SYSTEM OPC_Test
  (* Description: Showing how to use more than one forte on the same PC connection via OPC UA. One forte PC using as server, the other(s) as client(s). requirements: - one running forte PC on standard configuration - one running forte PC started on port 61599 ("-c localhost:61599") - OPC UA is required for all forte PCs *)
  (* Version 1.0, 2022-04-26, Maximilian Scharf *)
  APPLICATION OPC_TestApp
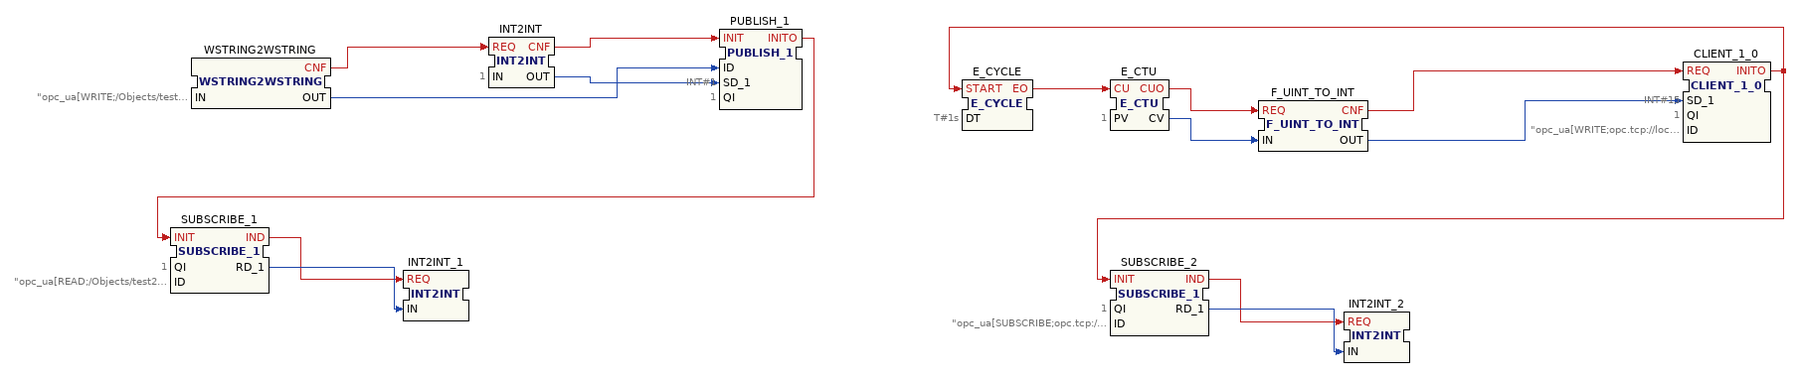
    (* Group __Group01: OPC UA documentation &#10;https://www.eclipse.org/4diac/en_help.php?helppage=html/communication/opc_ua_version1.html#build *)
    (* Group __Group02: OPC UA Server &#10;use: publish (WRITE) and subscribe (READ) *)
    (* Group __Group03: OPC UA Client &#10;use: client (WRITE) or subscribe (SUBSCRIBE) FBs *)
    (* Group __Group04: Use UaExpert Client for OPC UA connection and monitoring. *)
    FBS
      WSTRING2WSTRING : WSTRING2WSTRING(IN := "opc_ua[WRITE;/Objects/test1]"); {SET_ATTRIBUTE(GroupName, __Group02)}
      E_CTU : E_CTU(PV := 1); {SET_ATTRIBUTE(GroupName, __Group03)}
      E_CYCLE : E_CYCLE(DT := T#1s); {SET_ATTRIBUTE(GroupName, __Group03)}
      PUBLISH_1 : PUBLISH_1(QI := 1, SD_1 := INT#1); {SET_ATTRIBUTE(GroupName, __Group02)}
      CLIENT_1_0 : CLIENT_1_0(QI := 1, ID := "opc_ua[WRITE;opc.tcp://localhost:4840#;/Objects/test2]", SD_1 := INT#15); {SET_ATTRIBUTE(GroupName, __Group03)}
      INT2INT : INT2INT(IN := 1); {SET_ATTRIBUTE(GroupName, __Group02)}
      F_UINT_TO_INT : F_UINT_TO_INT; {SET_ATTRIBUTE(GroupName, __Group03)}
      SUBSCRIBE_1 : SUBSCRIBE_1(QI := 1, ID := "opc_ua[READ;/Objects/test2]"); {SET_ATTRIBUTE(GroupName, __Group02)}
      INT2INT_1 : INT2INT; {SET_ATTRIBUTE(GroupName, __Group02)}
      SUBSCRIBE_2 : SUBSCRIBE_1(QI := 1, ID := "opc_ua[SUBSCRIBE;opc.tcp://localhost:4840#;/Objects/test2]"); {SET_ATTRIBUTE(GroupName, __Group03)}
      INT2INT_2 : INT2INT; {SET_ATTRIBUTE(GroupName, __Group03)}
    END_FBS
    EVENT_CONNECTIONS
      E_CYCLE.EO TO E_CTU.CU;
      CLIENT_1_0.INITO TO E_CYCLE.START;
      INT2INT.CNF TO PUBLISH_1.INIT;
      WSTRING2WSTRING.CNF TO INT2INT.REQ;
      E_CTU.CUO TO F_UINT_TO_INT.REQ;
      F_UINT_TO_INT.CNF TO CLIENT_1_0.REQ;
      PUBLISH_1.INITO TO SUBSCRIBE_1.INIT;
      SUBSCRIBE_1.IND TO INT2INT_1.REQ;
      SUBSCRIBE_2.IND TO INT2INT_2.REQ;
      CLIENT_1_0.INITO TO SUBSCRIBE_2.INIT;
    END_CONNECTIONS
    DATA_CONNECTIONS
      WSTRING2WSTRING.OUT TO PUBLISH_1.ID;
      INT2INT.OUT TO PUBLISH_1.SD_1;
      E_CTU.CV TO F_UINT_TO_INT.IN;
      F_UINT_TO_INT.OUT TO CLIENT_1_0.SD_1;
      SUBSCRIBE_1.RD_1 TO INT2INT_1.IN;
      SUBSCRIBE_2.RD_1 TO INT2INT_2.IN;
    END_CONNECTIONS
  END_APPLICATION
  DEVICE Server : FORTE_PC(MGR_ID := "localhost:61498")
    {SET_ATTRIBUTE(Profile, DynamicTypeLoad)}
    {SET_ATTRIBUTE(FBType, GEN_E_MUX, F_LT, F_LWORD_TO_WORD, F_TAN, F_DINT_TO_UINT, F_BYTE_TO_DINT, F_ADD_DT_TIME, F_TIME_IN_US_TO_LREAL, F_INT_TO_UDINT, F_ADD_TOD_TIME, F_SUB_DT_DT, F_DT_TO_TOD, F_WSTRING_TO_REAL, F_UINT_TO_BCD_WORD, F_UDINT_TO_REAL, F_REAL_TO_UDINT, F_DWORD_TO_WORD, F_MUL, FB_CTUD_LINT, TEST_CONDITION, F_LE, GEN_SUBSCRIBE, F_LN, FB_CTD_DINT, GEN_OR, E_CYCLE, FB_F_TRIG, F_LREAL_TO_SINT, E_F_TRIG, F_LWORD_TO_UINT, E_RS, F_UINT_TO_WORD, F_WORD_TO_DINT, F_OR, F_WORD_TO_BYTE, F_TIME_IN_NS_TO_ULINT, FB_CTD_ULINT, FB_TOF, STEST_END, F_NE, FB_TON, F_STRING_TO_UINT, F_LWORD_TO_ULINT, F_INT_TO_STRING, F_INT_TO_BYTE, F_INT_TO_DINT, F_ULINT_TO_LINT, F_DWORD_TO_UINT, F_WSTRING_TO_ULINT, F_WSTRING_TO_LWORD, F_STRING_TO_DWORD, DWORD2DWORD, F_TIME_IN_NS_TO_LINT, F_DINT_TO_WSTRING, E_SELECT, F_LINT_TO_STRING, FB_CTUD, F_MULTIME, F_USINT_TO_INT, LocalizedText2LocalizedText, F_DWORD_TO_UDINT, F_UINT_TO_LWORD, F_SINT_TO_LWORD, GEN_F_MUX, USINT2USINT, F_LINT_TO_SINT, F_WORD_TO_USINT, F_DWORD_TO_INT, F_LREAL_TO_REAL, F_BOOL_TO_LINT, F_LEFT, FB_CTD, E_SR, F_UDINT_TO_BCD_DWORD, GEN_XOR, F_DINT_TO_WORD, F_SUB_TOD_TIME, E_RESTART, E_PERMIT, TIME2TIME, F_UINT_TO_SINT, F_XOR, F_STRING_TO_WORD, F_SEL, F_ULINT_TO_LREAL, F_SINT_TO_LREAL, F_DINT_TO_SINT, E_TimeOut, F_BYTE_TO_UDINT, F_REPLACE, F_LINT_TO_USINT, F_ABS, F_WORD_TO_LWORD, E_DELAY, GEN_ADD, F_INT_TO_WSTRING, F_STRING_TO_ULINT, F_USINT_TO_STRING, F_DINT_TO_USINT, F_STRING_TO_BOOL, F_DWORD_TO_WSTRING, F_INT_TO_REAL, F_DWORD_TO_STRING, E_CTU, F_TIME_TO_STRING, F_WSTRING_TO_BYTE, F_USINT_TO_WSTRING, F_WSTRING_TO_DINT, F_WSTRING_TO_DWORD, F_MOVE, F_WSTRING_TO_STRING, F_USINT_TO_LINT, F_DIV, F_WSTRING_TO_SINT, E_CTD, F_UINT_TO_DWORD, F_LWORD_TO_LINT, F_STRING_TO_TIME, FB_CTUD_DINT, F_ADD, F_BYTE_TO_LINT, F_TIME_IN_MS_TO_LREAL, F_LREAL_TO_UINT, F_ACOS, F_DWORD_TO_LINT, F_SHL, F_REAL_TO_ULINT, F_ULINT_TO_UINT, F_UDINT_TO_SINT, F_SHR, F_BOOL_TO_INT, UINT2UINT, F_WORD_TO_DWORD, F_INT_TO_LWORD, F_USINT_TO_UINT, F_LREAL_TO_WSTRING, F_INT_TO_ULINT, GEN_CSV_WRITER, F_LINT_TO_WORD, F_UINT_TO_LREAL, F_STRING_TO_SINT, F_SINT_TO_WORD, F_STRING_TO_WSTRING, STRING2STRING, F_LREAL_TO_DINT, F_SIN, F_UINT_TO_USINT, FB_CTU_LINT, F_DINT_TO_ULINT, F_REAL_TO_UINT, RMT_RES, F_ULINT_TO_WORD, F_INT_TO_LINT, E_D_FF, F_STRING_TO_USINT, FB_CTD_LINT, FB_R_TRIG, F_INT_TO_DWORD, F_WORD_TO_LINT, F_UDINT_TO_INT, REAL2REAL, F_LREAL_TO_STRING, F_WSTRING_TO_INT, F_LREAL_TO_USINT, F_DINT_TO_LWORD, DEV_MGR, F_SINT_TO_UINT, E_CTUD, E_RDELAY, F_SINT_TO_ULINT, F_LINT_TO_ULINT, F_RIGHT, F_SINT_TO_INT, F_LWORD_TO_WSTRING, SINT2SINT, FB_CTD_UDINT, F_LINT_TO_LWORD, F_LWORD_TO_UDINT, F_LWORD_TO_STRING, F_TRUNC, F_ULINT_TO_DWORD, F_TIME_IN_S_TO_LREAL, F_BOOL_TO_DWORD, E_TRAIN, OUT_ANY_CONSOLE, F_ULINT_TO_SINT, F_DINT_TO_LINT, F_BOOL_TO_USINT, F_UDINT_TO_DWORD, GEN_E_DEMUX, F_SQRT, F_BOOL_TO_DINT, F_BOOL_TO_BYTE, F_UINT_TO_INT, F_TIME_IN_S_TO_LINT, F_ULINT_TO_USINT, F_UINT_TO_REAL, F_LREAL_TO_LWORD, F_SINT_TO_LINT, F_MAX, F_LREAL_TO_INT, F_UDINT_TO_LWORD, INT2INT, F_BYTE_TO_ULINT, F_UDINT_TO_WORD, F_LINT_TO_UINT, F_TIME_IN_US_TO_ULINT, F_COS, F_TIME_IN_NS_TO_LREAL, F_REAL_TO_LINT, F_STRING_TO_LWORD, F_BYTE_TO_STRING, F_USINT_TO_WORD, E_REND, F_ASIN, F_REAL_TO_INT, F_BOOL_TO_LWORD, F_WORD_BCD_TO_UINT, F_BOOL_TO_SINT, F_BYTE_TO_INT, F_BOOL_TO_ULINT, EMB_RES, F_BYTE_TO_WORD, F_STRING_TO_INT, F_USINT_TO_LWORD, F_DWORD_TO_DINT, F_ULINT_TO_LWORD, GEN_APPEND_STRING, F_USINT_TO_ULINT, GEN_SUBL, F_DWORD_TO_BYTE, F_DIVTIME, F_ROL, F_LWORD_TO_DINT, F_WORD_TO_SINT, F_STRING_TO_REAL, F_LWORD_TO_BYTE, FB_CTU_DINT, GEN_AND, F_AND, F_ROR, GEN_CLIENT, F_ULINT_TO_WSTRING, F_SINT_TO_STRING, F_LREAL_TO_LINT, WSTRING2WSTRING, F_WORD_TO_INT, F_UINT_TO_BYTE, F_UDINT_TO_UINT, F_SINT_TO_UDINT, F_UINT_TO_DINT, F_UINT_TO_UDINT, F_UINT_TO_WSTRING, F_WSTRING_TO_UINT, F_DINT_TO_UDINT, E_SPLIT, F_DWORD_TO_LWORD, F_USINT_TO_SINT, F_ULINT_TO_BCD_LWORD, F_BYTE_BCD_TO_USINT, F_DWORD_TO_ULINT, F_BYTE_TO_SINT, F_BYTE_TO_WSTRING, GEN_ARRAY2ARRAY, F_DT_TO_DATE, GEN_STRUCT_DEMUX, F_LEN, GEN_STRUCT_MUX, F_INT_TO_WORD, FB_RANDOM, F_LINT_TO_UDINT, F_EXP, F_USINT_TO_DWORD, F_TIME_IN_MS_TO_ULINT, F_REAL_TO_SINT, F_INT_TO_USINT, F_UDINT_TO_WSTRING, F_EXPT, F_SUB, F_ULINT_TO_REAL, F_REAL_TO_LREAL, F_MID, F_BYTE_TO_UINT, F_BYTE_TO_DWORD, F_INT_TO_UINT, F_DWORD_TO_REAL, F_DINT_TO_BYTE, F_WORD_TO_STRING, F_REAL_TO_STRING, F_SUB_TOD_TOD, SET_AT_INDEX, F_MIN, F_LREAL_TO_ULINT, F_STRING_TO_BYTE, F_BYTE_TO_LWORD, F_STRING_TO_DINT, F_WORD_TO_WSTRING, BOOL2BOOL, F_LINT_TO_INT, F_WSTRING_TO_TIME, FB_CTU_UDINT, F_WSTRING_TO_BOOL, F_INSERT, F_SUB_DT_TIME, F_FIND, F_UDINT_TO_ULINT, F_WORD_TO_UDINT, F_DINT_TO_DWORD, F_WSTRING_TO_USINT, GEN_VALUES2ARRAY, GEN_ARRAY2VALUES, F_WSTRING_TO_WORD, F_DINT_TO_STRING, F_WORD_TO_UINT, F_TIME_IN_US_TO_LINT, F_LINT_TO_DWORD, F_CONCAT, FB_CTUD_ULINT, F_UDINT_TO_LINT, F_SUB_DATE_DATE, F_LWORD_TO_LREAL, F_LWORD_TO_INT, WORD2WORD, E_STOPWATCH, F_LIMIT, F_TIME_IN_S_TO_ULINT, F_LWORD_TO_USINT, F_REAL_TO_DINT, F_DWORD_TO_USINT, E_MERGE, F_SINT_TO_DWORD, E_DEMUX, F_BOOL_TO_UDINT, BYTE2BYTE, FB_TP, F_USINT_TO_BCD_BYTE, F_SINT_TO_DINT, F_UINT_TO_LINT, F_SINT_TO_BYTE, F_ATAN, F_LINT_TO_BYTE, F_BYTE_TO_USINT, F_ULINT_TO_UDINT, FB_SR, F_NOT, F_DINT_TO_INT, F_LINT_TO_DINT, F_DELETE, FB_CTU, GEN_SERVER, GEN_PUBL, F_UDINT_TO_LREAL, F_BOOL_TO_UINT, F_UINT_TO_STRING, E_R_TRIG, F_GE, F_LWORD_BCD_TO_ULINT, F_UDINT_TO_STRING, F_REAL_TO_WSTRING, FB_RS, F_MUX_2, F_LINT_TO_WSTRING, F_USINT_TO_UDINT, F_UINT_TO_ULINT, F_EQ, E_T_FF, F_USINT_TO_REAL, LREAL2LREAL, F_STRING_TO_LREAL, F_ULINT_TO_STRING, F_MOD, E_RTimeOut, F_ULINT_TO_DINT, F_ULINT_TO_BYTE, F_WSTRING_TO_UDINT, F_TIME_TO_WSTRING, GET_STRUCT_VALUE, GEN_PUBLISH, F_REAL_TO_DWORD, F_DWORD_BCD_TO_UDINT, F_INT_TO_LREAL, F_SINT_TO_WSTRING, F_LWORD_TO_SINT, F_GT, F_LINT_TO_REAL, F_TIME_IN_MS_TO_LINT, F_SINT_TO_REAL, F_LOG, F_ULINT_TO_INT, F_DWORD_TO_SINT, F_BOOL_TO_WORD, F_REAL_TO_USINT, E_SWITCH, F_LINT_TO_LREAL, F_STRING_TO_LINT, F_SINT_TO_USINT, F_DINT_TO_REAL, DINT2DINT, F_WORD_TO_ULINT, F_INT_TO_SINT, F_CONCAT_DATE_TOD, F_WSTRING_TO_LREAL, GET_AT_INDEX, F_USINT_TO_LREAL, F_BOOL_TO_WSTRING, FB_CTU_ULINT, F_DINT_TO_LREAL, UDINT2UDINT, F_USINT_TO_BYTE, F_BOOL_TO_STRING, F_LWORD_TO_DWORD, F_LREAL_TO_UDINT, F_STRING_TO_UDINT, F_UDINT_TO_DINT, F_UDINT_TO_BYTE, F_WSTRING_TO_LINT, F_USINT_TO_DINT)} (* created during deployment *)
    RESOURCE EMB_RES : EMB_RES
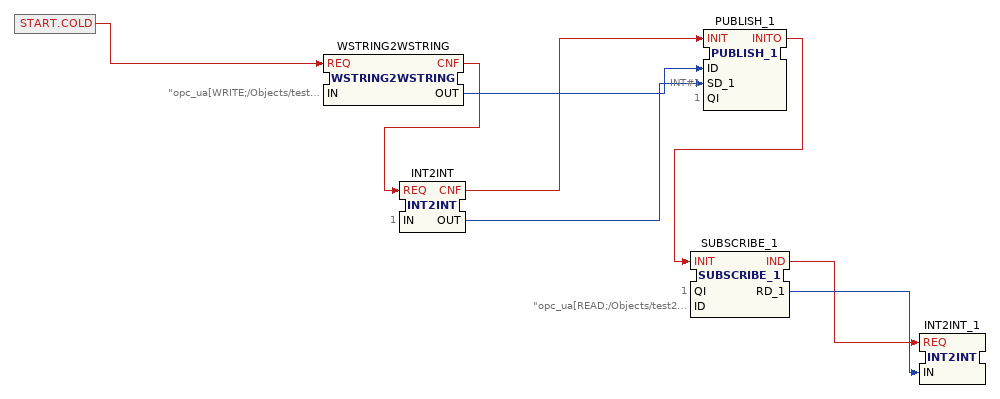
      FBS
        WSTRING2WSTRING : WSTRING2WSTRING(IN := "opc_ua[WRITE;/Objects/test1]");
        PUBLISH_1 : PUBLISH_1(QI := 1, SD_1 := INT#1);
        INT2INT : INT2INT(IN := 1);
        SUBSCRIBE_1 : SUBSCRIBE_1(QI := 1, ID := "opc_ua[READ;/Objects/test2]");
        INT2INT_1 : INT2INT;
      END_FBS
      EVENT_CONNECTIONS
        START.COLD TO WSTRING2WSTRING.REQ;
        INT2INT.CNF TO PUBLISH_1.INIT;
        WSTRING2WSTRING.CNF TO INT2INT.REQ;
        PUBLISH_1.INITO TO SUBSCRIBE_1.INIT;
        SUBSCRIBE_1.IND TO INT2INT_1.REQ;
      END_CONNECTIONS
      DATA_CONNECTIONS
        WSTRING2WSTRING.OUT TO PUBLISH_1.ID;
        INT2INT.OUT TO PUBLISH_1.SD_1;
        SUBSCRIBE_1.RD_1 TO INT2INT_1.IN;
      END_CONNECTIONS
    END_RESOURCE
  END_DEVICE
  DEVICE Client : FORTE_PC(MGR_ID := "localhost:61497")
    {SET_ATTRIBUTE(Profile, DynamicTypeLoad)}
    {SET_ATTRIBUTE(FBType, GEN_E_MUX, F_LT, F_LWORD_TO_WORD, F_TAN, F_DINT_TO_UINT, F_BYTE_TO_DINT, F_ADD_DT_TIME, F_TIME_IN_US_TO_LREAL, F_INT_TO_UDINT, F_ADD_TOD_TIME, F_SUB_DT_DT, F_DT_TO_TOD, F_WSTRING_TO_REAL, F_UINT_TO_BCD_WORD, F_UDINT_TO_REAL, F_REAL_TO_UDINT, F_DWORD_TO_WORD, F_MUL, FB_CTUD_LINT, TEST_CONDITION, F_LE, GEN_SUBSCRIBE, F_LN, FB_CTD_DINT, GEN_OR, E_CYCLE, FB_F_TRIG, F_LREAL_TO_SINT, E_F_TRIG, F_LWORD_TO_UINT, E_RS, F_UINT_TO_WORD, F_WORD_TO_DINT, F_OR, F_WORD_TO_BYTE, F_TIME_IN_NS_TO_ULINT, FB_CTD_ULINT, FB_TOF, STEST_END, F_NE, FB_TON, F_STRING_TO_UINT, F_LWORD_TO_ULINT, F_INT_TO_STRING, F_INT_TO_BYTE, F_INT_TO_DINT, F_ULINT_TO_LINT, F_DWORD_TO_UINT, F_WSTRING_TO_ULINT, F_WSTRING_TO_LWORD, F_STRING_TO_DWORD, DWORD2DWORD, F_TIME_IN_NS_TO_LINT, F_DINT_TO_WSTRING, E_SELECT, F_LINT_TO_STRING, FB_CTUD, F_MULTIME, F_USINT_TO_INT, LocalizedText2LocalizedText, F_DWORD_TO_UDINT, F_UINT_TO_LWORD, F_SINT_TO_LWORD, GEN_F_MUX, USINT2USINT, F_LINT_TO_SINT, F_WORD_TO_USINT, F_DWORD_TO_INT, F_LREAL_TO_REAL, F_BOOL_TO_LINT, F_LEFT, FB_CTD, E_SR, F_UDINT_TO_BCD_DWORD, GEN_XOR, F_DINT_TO_WORD, F_SUB_TOD_TIME, E_RESTART, E_PERMIT, TIME2TIME, F_UINT_TO_SINT, F_XOR, F_STRING_TO_WORD, F_SEL, F_ULINT_TO_LREAL, F_SINT_TO_LREAL, F_DINT_TO_SINT, E_TimeOut, F_BYTE_TO_UDINT, F_REPLACE, F_LINT_TO_USINT, F_ABS, F_WORD_TO_LWORD, E_DELAY, GEN_ADD, F_INT_TO_WSTRING, F_STRING_TO_ULINT, F_USINT_TO_STRING, F_DINT_TO_USINT, F_STRING_TO_BOOL, F_DWORD_TO_WSTRING, F_INT_TO_REAL, F_DWORD_TO_STRING, E_CTU, F_TIME_TO_STRING, F_WSTRING_TO_BYTE, F_USINT_TO_WSTRING, F_WSTRING_TO_DINT, F_WSTRING_TO_DWORD, F_MOVE, F_WSTRING_TO_STRING, F_USINT_TO_LINT, F_DIV, F_WSTRING_TO_SINT, E_CTD, F_UINT_TO_DWORD, F_LWORD_TO_LINT, F_STRING_TO_TIME, FB_CTUD_DINT, F_ADD, F_BYTE_TO_LINT, F_TIME_IN_MS_TO_LREAL, F_LREAL_TO_UINT, F_ACOS, F_DWORD_TO_LINT, F_SHL, F_REAL_TO_ULINT, F_ULINT_TO_UINT, F_UDINT_TO_SINT, F_SHR, F_BOOL_TO_INT, UINT2UINT, F_WORD_TO_DWORD, F_INT_TO_LWORD, F_USINT_TO_UINT, F_LREAL_TO_WSTRING, F_INT_TO_ULINT, GEN_CSV_WRITER, F_LINT_TO_WORD, F_UINT_TO_LREAL, F_STRING_TO_SINT, F_SINT_TO_WORD, F_STRING_TO_WSTRING, STRING2STRING, F_LREAL_TO_DINT, F_SIN, F_UINT_TO_USINT, FB_CTU_LINT, F_DINT_TO_ULINT, F_REAL_TO_UINT, RMT_RES, F_ULINT_TO_WORD, F_INT_TO_LINT, E_D_FF, F_STRING_TO_USINT, FB_CTD_LINT, FB_R_TRIG, F_INT_TO_DWORD, F_WORD_TO_LINT, F_UDINT_TO_INT, REAL2REAL, F_LREAL_TO_STRING, F_WSTRING_TO_INT, F_LREAL_TO_USINT, F_DINT_TO_LWORD, DEV_MGR, F_SINT_TO_UINT, E_CTUD, E_RDELAY, F_SINT_TO_ULINT, F_LINT_TO_ULINT, F_RIGHT, F_SINT_TO_INT, F_LWORD_TO_WSTRING, SINT2SINT, FB_CTD_UDINT, F_LINT_TO_LWORD, F_LWORD_TO_UDINT, F_LWORD_TO_STRING, F_TRUNC, F_ULINT_TO_DWORD, F_TIME_IN_S_TO_LREAL, F_BOOL_TO_DWORD, E_TRAIN, OUT_ANY_CONSOLE, F_ULINT_TO_SINT, F_DINT_TO_LINT, F_BOOL_TO_USINT, F_UDINT_TO_DWORD, GEN_E_DEMUX, F_SQRT, F_BOOL_TO_DINT, F_BOOL_TO_BYTE, F_UINT_TO_INT, F_TIME_IN_S_TO_LINT, F_ULINT_TO_USINT, F_UINT_TO_REAL, F_LREAL_TO_LWORD, F_SINT_TO_LINT, F_MAX, F_LREAL_TO_INT, F_UDINT_TO_LWORD, INT2INT, F_BYTE_TO_ULINT, F_UDINT_TO_WORD, F_LINT_TO_UINT, F_TIME_IN_US_TO_ULINT, F_COS, F_TIME_IN_NS_TO_LREAL, F_REAL_TO_LINT, F_STRING_TO_LWORD, F_BYTE_TO_STRING, F_USINT_TO_WORD, E_REND, F_ASIN, F_REAL_TO_INT, F_BOOL_TO_LWORD, F_WORD_BCD_TO_UINT, F_BOOL_TO_SINT, F_BYTE_TO_INT, F_BOOL_TO_ULINT, EMB_RES, F_BYTE_TO_WORD, F_STRING_TO_INT, F_USINT_TO_LWORD, F_DWORD_TO_DINT, F_ULINT_TO_LWORD, GEN_APPEND_STRING, F_USINT_TO_ULINT, GEN_SUBL, F_DWORD_TO_BYTE, F_DIVTIME, F_ROL, F_LWORD_TO_DINT, F_WORD_TO_SINT, F_STRING_TO_REAL, F_LWORD_TO_BYTE, FB_CTU_DINT, GEN_AND, F_AND, F_ROR, GEN_CLIENT, F_ULINT_TO_WSTRING, F_SINT_TO_STRING, F_LREAL_TO_LINT, WSTRING2WSTRING, F_WORD_TO_INT, F_UINT_TO_BYTE, F_UDINT_TO_UINT, F_SINT_TO_UDINT, F_UINT_TO_DINT, F_UINT_TO_UDINT, F_UINT_TO_WSTRING, F_WSTRING_TO_UINT, F_DINT_TO_UDINT, E_SPLIT, F_DWORD_TO_LWORD, F_USINT_TO_SINT, F_ULINT_TO_BCD_LWORD, F_BYTE_BCD_TO_USINT, F_DWORD_TO_ULINT, F_BYTE_TO_SINT, F_BYTE_TO_WSTRING, GEN_ARRAY2ARRAY, F_DT_TO_DATE, GEN_STRUCT_DEMUX, F_LEN, GEN_STRUCT_MUX, F_INT_TO_WORD, FB_RANDOM, F_LINT_TO_UDINT, F_EXP, F_USINT_TO_DWORD, F_TIME_IN_MS_TO_ULINT, F_REAL_TO_SINT, F_INT_TO_USINT, F_UDINT_TO_WSTRING, F_EXPT, F_SUB, F_ULINT_TO_REAL, F_REAL_TO_LREAL, F_MID, F_BYTE_TO_UINT, F_BYTE_TO_DWORD, F_INT_TO_UINT, F_DWORD_TO_REAL, F_DINT_TO_BYTE, F_WORD_TO_STRING, F_REAL_TO_STRING, F_SUB_TOD_TOD, SET_AT_INDEX, F_MIN, F_LREAL_TO_ULINT, F_STRING_TO_BYTE, F_BYTE_TO_LWORD, F_STRING_TO_DINT, F_WORD_TO_WSTRING, BOOL2BOOL, F_LINT_TO_INT, F_WSTRING_TO_TIME, FB_CTU_UDINT, F_WSTRING_TO_BOOL, F_INSERT, F_SUB_DT_TIME, F_FIND, F_UDINT_TO_ULINT, F_WORD_TO_UDINT, F_DINT_TO_DWORD, F_WSTRING_TO_USINT, GEN_VALUES2ARRAY, GEN_ARRAY2VALUES, F_WSTRING_TO_WORD, F_DINT_TO_STRING, F_WORD_TO_UINT, F_TIME_IN_US_TO_LINT, F_LINT_TO_DWORD, F_CONCAT, FB_CTUD_ULINT, F_UDINT_TO_LINT, F_SUB_DATE_DATE, F_LWORD_TO_LREAL, F_LWORD_TO_INT, WORD2WORD, E_STOPWATCH, F_LIMIT, F_TIME_IN_S_TO_ULINT, F_LWORD_TO_USINT, F_REAL_TO_DINT, F_DWORD_TO_USINT, E_MERGE, F_SINT_TO_DWORD, E_DEMUX, F_BOOL_TO_UDINT, BYTE2BYTE, FB_TP, F_USINT_TO_BCD_BYTE, F_SINT_TO_DINT, F_UINT_TO_LINT, F_SINT_TO_BYTE, F_ATAN, F_LINT_TO_BYTE, F_BYTE_TO_USINT, F_ULINT_TO_UDINT, FB_SR, F_NOT, F_DINT_TO_INT, F_LINT_TO_DINT, F_DELETE, FB_CTU, GEN_SERVER, GEN_PUBL, F_UDINT_TO_LREAL, F_BOOL_TO_UINT, F_UINT_TO_STRING, E_R_TRIG, F_GE, F_LWORD_BCD_TO_ULINT, F_UDINT_TO_STRING, F_REAL_TO_WSTRING, FB_RS, F_MUX_2, F_LINT_TO_WSTRING, F_USINT_TO_UDINT, F_UINT_TO_ULINT, F_EQ, E_T_FF, F_USINT_TO_REAL, LREAL2LREAL, F_STRING_TO_LREAL, F_ULINT_TO_STRING, F_MOD, E_RTimeOut, F_ULINT_TO_DINT, F_ULINT_TO_BYTE, F_WSTRING_TO_UDINT, F_TIME_TO_WSTRING, GET_STRUCT_VALUE, GEN_PUBLISH, F_REAL_TO_DWORD, F_DWORD_BCD_TO_UDINT, F_INT_TO_LREAL, F_SINT_TO_WSTRING, F_LWORD_TO_SINT, F_GT, F_LINT_TO_REAL, F_TIME_IN_MS_TO_LINT, F_SINT_TO_REAL, F_LOG, F_ULINT_TO_INT, F_DWORD_TO_SINT, F_BOOL_TO_WORD, F_REAL_TO_USINT, E_SWITCH, F_LINT_TO_LREAL, F_STRING_TO_LINT, F_SINT_TO_USINT, F_DINT_TO_REAL, DINT2DINT, F_WORD_TO_ULINT, F_INT_TO_SINT, F_CONCAT_DATE_TOD, F_WSTRING_TO_LREAL, GET_AT_INDEX, F_USINT_TO_LREAL, F_BOOL_TO_WSTRING, FB_CTU_ULINT, F_DINT_TO_LREAL, UDINT2UDINT, F_USINT_TO_BYTE, F_BOOL_TO_STRING, F_LWORD_TO_DWORD, F_LREAL_TO_UDINT, F_STRING_TO_UDINT, F_UDINT_TO_DINT, F_UDINT_TO_BYTE, F_WSTRING_TO_LINT, F_USINT_TO_DINT)} (* created during deployment *)
    RESOURCE EMB_RES : EMB_RES
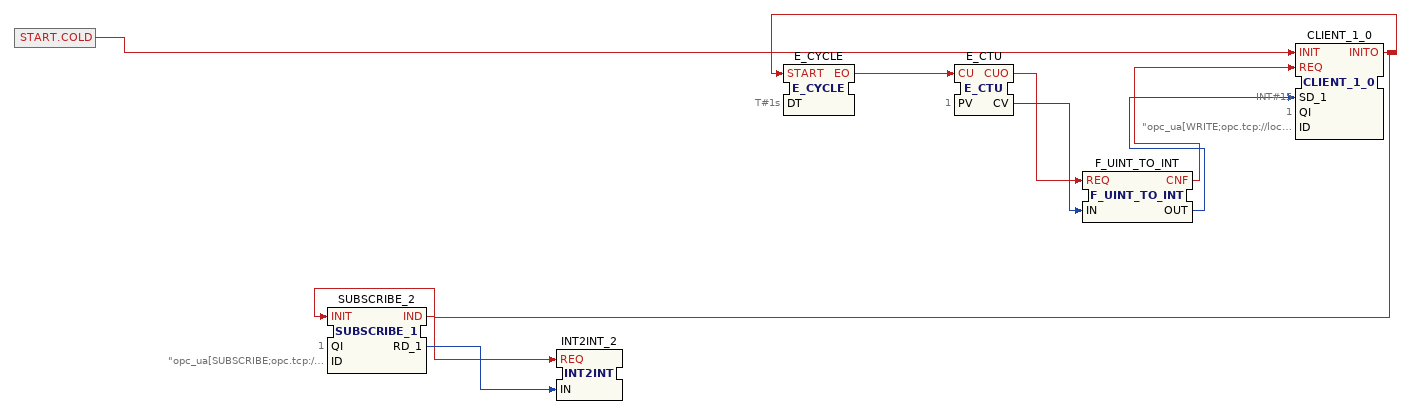
      FBS
        E_CTU : E_CTU(PV := 1);
        E_CYCLE : E_CYCLE(DT := T#1s);
        CLIENT_1_0 : CLIENT_1_0(QI := 1, ID := "opc_ua[WRITE;opc.tcp://localhost:4840#;/Objects/test2]", SD_1 := INT#15);
        F_UINT_TO_INT : F_UINT_TO_INT;
        INT2INT_2 : INT2INT;
        SUBSCRIBE_2 : SUBSCRIBE_1(QI := 1, ID := "opc_ua[SUBSCRIBE;opc.tcp://localhost:4840#;/Objects/test2]");
      END_FBS
      EVENT_CONNECTIONS
        E_CYCLE.EO TO E_CTU.CU;
        CLIENT_1_0.INITO TO E_CYCLE.START;
        START.COLD TO CLIENT_1_0.INIT;
        E_CTU.CUO TO F_UINT_TO_INT.REQ;
        F_UINT_TO_INT.CNF TO CLIENT_1_0.REQ;
        CLIENT_1_0.INITO TO SUBSCRIBE_2.INIT;
        SUBSCRIBE_2.IND TO INT2INT_2.REQ;
      END_CONNECTIONS
      DATA_CONNECTIONS
        E_CTU.CV TO F_UINT_TO_INT.IN;
        F_UINT_TO_INT.OUT TO CLIENT_1_0.SD_1;
        SUBSCRIBE_2.RD_1 TO INT2INT_2.IN;
      END_CONNECTIONS
    END_RESOURCE
  END_DEVICE
  MAPPINGS
    OPC_TestApp.WSTRING2WSTRING ON Server.EMB_RES.WSTRING2WSTRING;
    OPC_TestApp.E_CTU ON Client.EMB_RES.E_CTU;
    OPC_TestApp.E_CYCLE ON Client.EMB_RES.E_CYCLE;
    OPC_TestApp.PUBLISH_1 ON Server.EMB_RES.PUBLISH_1;
    OPC_TestApp.CLIENT_1_0 ON Client.EMB_RES.CLIENT_1_0;
    OPC_TestApp.INT2INT ON Server.EMB_RES.INT2INT;
    OPC_TestApp.F_UINT_TO_INT ON Client.EMB_RES.F_UINT_TO_INT;
    OPC_TestApp.SUBSCRIBE_1 ON Server.EMB_RES.SUBSCRIBE_1;
    OPC_TestApp.INT2INT_1 ON Server.EMB_RES.INT2INT_1;
    OPC_TestApp.INT2INT_2 ON Client.EMB_RES.INT2INT_2;
    OPC_TestApp.SUBSCRIBE_2 ON Client.EMB_RES.SUBSCRIBE_2;
  END_MAPPINGS
END_SYSTEM
